// Mitsubishi GX Works2 project: LRI - PLC - NAND   PLC: Q03UDV

PROGRAM MAIN
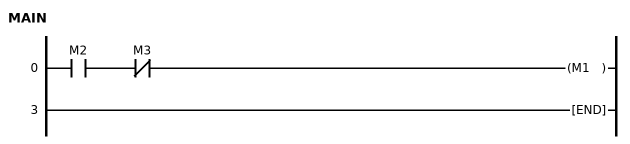
0     LD      M2
      ANI     M3
      OUT     M1
3     END
END_PROGRAM
